Yaskawa INFORM job: FUUUUU.JBI

/JOB
//NAME FUUUUU
//POS
///NPOS 4,0,0,0
///TOOL 0
///PULSE
C000=30334,49152,-58316,3555,4172,9939
C001=7167,49725,-55876,3555,3624,9786
C002=-2945,48206,-38174,3555,1738,9261
C003=-19010,40224,-24764,3555,-1260,8427
//INST
///DATE 2014/09/13 21:44
///ATTR 0,0,0,0,0,0,0,0,0,0,0,0,0,1,0,0
///FRAME BASE
NOP
*U
MOVJ C000 VJ=50.00 CONT
MOVJ C001 VJ=75.00 CONT
MOVJ C002 VJ=100.00 CONT
MOVJ C003 VJ=50.00 CONT
JUMP *U
END
